TYPE
    TcoComprehensiveResult :
    STRUCT
		{attribute addProperty  Name "<#Result#>"}
        Result     : eOverallResult;
		{attribute addProperty  Name "<#Failures#>"}
        Failures   : STRING(255);
		{attribute addProperty  Name "<#ErrorCodes#>"}
        ErrorCodes : STRING(255);
    END_STRUCT
END_TYPE

(* stored: Version 1.1.0.1, ProductVersion 3.1.4024.12
   DUT TcoComprehensiveResult: Id {a33ed128-190c-09d3-3fba-9a17f28b94b9} *)
